INTERFACE I_ConvertUnitsLREAL EXTENDS I_Fallible


METHOD ConvertQuantityLREAL
VAR_INPUT
	QuantityToConvert : I_QuantityLREAL;
	DesiredUnits : T_MaxString;
END_VAR
VAR_IN_OUT
    ConvertedQuantity : FB_QuantityLREALPublic(Units := '1');
END_VAR
END_METHOD

END_INTERFACE

(* stored: Version 1.1.0.1
   Itf I_ConvertUnitsLREAL: Id {55f893e7-7529-4e2a-810b-ffc51e01748c}
   Method ConvertQuantityLREAL: Id {8c4614a7-f27b-4200-8c1b-600b2d2f5c07} *)
